(* Logix 5000 project; controller HP_SSC01 vendor 1 type 14 code 67 rev 17.7; software revision 17.01; part 8 of 15 *)
(* tags used below, declared in another part *)
   A_C3_0300 : ALIAS FOR C3_FaultStandard.0;
   A_C3_0301 : ALIAS FOR C3_FaultStandard.1;
   A_C3_0302 : ALIAS FOR C3_FaultStandard.2;
   A_C3_0303 : ALIAS FOR C3_FaultStandard.3;
   A_C3_0305 : ALIAS FOR C3_FaultStandard.5;
   A_C3_0309 : ALIAS FOR C3_FaultStandard.9;
   A_C3_0310 : ALIAS FOR C3_FaultStandard.10;
   A_C3_0311 : ALIAS FOR C3_FaultStandard.11;
   A_C3_0312 : ALIAS FOR C3_FaultStandard.12;
   A_C3_0313 : ALIAS FOR C3_FaultStandard.13;
   A_C3_0314 : ALIAS FOR C3_FaultStandard.14;
   A_C3_0315 : ALIAS FOR C3_FaultStandard.15;
   A_C3_0317 : ALIAS FOR C3_FaultStandard.17;
   A_C3_0319 : ALIAS FOR C3_FaultStandard.19;
   A_C3_0321 : ALIAS FOR C3_FaultStandard.21;
   A_C3_0322 : ALIAS FOR C3_FaultStandard.22;
   A_C3_0323 : ALIAS FOR C3_FaultStandard.23;
   A_C3_0324 : ALIAS FOR C3_FaultStandard.24;
   A_C3_0325 : ALIAS FOR C3_FaultStandard.25;
   A_C3_0327 : ALIAS FOR C3_FaultStandard.27;
   A_C3_0328 : ALIAS FOR C3_FaultStandard.28;
   A_C3_0329 : ALIAS FOR C3_FaultStandard.29;
   A_C3_0330 : ALIAS FOR C3_FaultStandard.30;
   A_C3_0331 : ALIAS FOR C3_FaultStandard.31;
   A_C3_0404 : ALIAS FOR C3_Warning.4;
   A_C3_0406 : ALIAS FOR C3_Warning.6;
   A_C3_0407 : ALIAS FOR C3_Warning.7;
   A_C3_0408 : ALIAS FOR C3_Warning.8;
   A_C3_0409 : ALIAS FOR C3_Warning.9;
   A_C3_0412 : ALIAS FOR C3_Warning.12;
   A_C3_0413 : ALIAS FOR C3_Warning.13;
   A_C3_0414 : ALIAS FOR C3_Warning.14;
   A_C3_0415 : ALIAS FOR C3_Warning.15;
   A_C3_0416 : ALIAS FOR C3_Warning.16;
   A_C3_0424 : ALIAS FOR C3_Warning.24;
   A_C3_0427 : ALIAS FOR C3_Warning.27;
   A_C3_0428 : ALIAS FOR C3_Warning.28;
   A_C3_0430 : ALIAS FOR C3_Warning.30;
   C3 : AXIS_SERVO_DRIVE;
   C3_32HourTimers : TIMER[4];
   C3_All_DLY_OK : BOOL;
   C3_BrakeSequenceInProcess : BOOL;
   C3_BrakeTest : BOOL;
   C3_BrakeTestEndPosition : REAL;
   C3_BrakeTestFailed : BOOL;
   C3_BrakeTestLocalDisable : BOOL;
   C3_BrakeTestMAJ01 : MOTION_INSTRUCTION;
   C3_BrakeTestMessageNumber : DINT;
   C3_BrakeTestONS : BOOL;
   C3_BrakeTestSelected : BOOL;
   C3_BrakeTestSequence : DINT;
   C3_BrakeTestSequenceAlarms : DINT;
   C3_BrakeTestSequenceAlarmTimer : TIMER[16];
   C3_BrakeTestSequenceONS : DINT;
   C3_BrakeTestStartPosition : REAL;
   C3_BrakeTestStoppingDistance : REAL;
   C3_BrakeTestTimerHoldVel : TIMER;
   C3_BrakeTestWarning : BOOL;
   C3_DisableTimer : TIMER;
   C3_DumpTest : BOOL;
   C3_DumpValveFailedOff : BOOL;
   C3_DumpValveFailedOn : BOOL;
   C3_DumpValveMessageNumber : DINT;
   C3_DumpValveTestDelay : TIMER[8];
   C3_DumpValveTestDelay2 : TIMER;
   C3_DumpValveTestSelected : BOOL;
   C3_DumpValveTestSequence : DINT;
   C3_DumpValveTestSequenceAlarms : DINT;
   C3_DumpValveTestSequenceAlarmTimer : TIMER[16];
   C3_EncoderCounts : DINT;
   C3_EncoderCountsRaw : ALIAS FOR C3_RIO_AENT:3:I.PresentData;
   C3_EncoderDegree : REAL;
   C3_FaultDebounce : TIMER[8];
   C3_FaultHoldTimer : TIMER[4];
   C3_FaultHomeSwitchNotFound : BOOL;
   C3_FaultStandard : DINT;
   C3_HomeInputStatus : BOOL;
   C3_HomeSequence : DINT;
   C3_HomeSequenceAlarms : DINT;
   C3_HomeSwitchFaultK7KFailedOff : BOOL;
   C3_HomeSwitchFaultK7KFailedOn : BOOL;
   C3_HomeSwitchFaultSafeFailedOff : BOOL;
   C3_HomeSwitchFaultSafeFailedOn : BOOL;
   C3_IndexEnable : BOOL;
   C3_JogEnable : BOOL;
   C3_LIM_ALARM_B : ALIAS FOR C3_RIO_AENT:I.Data[1].0;
   C3_MaintEnable : BOOL;
   C3_MotorActualPositionX1000 : DINT;
   C3_MotorAverageVelocityX1000 : DINT;
   C3_MotorFan : ALIAS FOR C3_RIO_AENT:O.Data[2].0;
   C3_MSF : MOTION_INSTRUCTION;
   C3_MSO : MOTION_INSTRUCTION;
   C3_OIT_Current : DINT;
   C3_ONS_Fault : DINT;
   C3_RemoteBrakeAndHomeSequenceAlarms : DINT;
   C3_RemoteBrakeTestCMD : BOOL;
   C3_RemoteDumpTestCMD : BOOL;
   C3_ServoActionStatusOffDelay : TIMER;
   C3_ServoActionStatusOnDelay : TIMER;
   C3_ServoFanOverload : ALIAS FOR C3_RIO_AENT:I.Data[1].2;
   C3_SS_LocalRemote_1_IsRemote : ALIAS FOR C3_RIO_AENT:1:I.3;
   C3_SS_RemoteMode : BOOL;
   C3_Warning : DINT;
   C3DumpValveTestSequenceONS : DINT;
   RCS_CMD_RunInAuto : BOOL;
   RCS_SyncMotionEnable : BOOL;
   S_C3_EncoderDegree : DINT;
   S_C3_ExecutePB : BOOL;
   S_C3_FaultReset : BOOL;
   S_C3_ModeLocal : BOOL;
   S_C3_ModeRemote : BOOL;
   S_C3_MotionEnabled : BOOL;
   S_C3_MSTOP_InputOK : BOOL;
   S_C3_NearOnPath : BOOL;
   S_C3_OffPath : BOOL;
   S_C3_OIT_FaultReset : BOOL;
   S_C3_OutputEnable : BOOL;
   S_C3_PressureOK : ALIAS FOR C3_Safe:I.Pt05Data;
   S_C3_SAFETY_ENABLE_1 : ALIAS FOR C3_Safe:O.Pt00Data;
   S_C3_SAFETY_ENABLE_2 : ALIAS FOR C3_Safe:O.Pt01Data;
   S_C3_Stop1_OK : BOOL;
   S_RCS_CMD_FaultReset : BOOL;
   STS_Enable_Rail : DINT;
   ZZZ_DIAG_A_C3_0302 : BOOL;
   ZZZ_DIAG_C3_AxisFault : DINT;
   ZZZ_DIAG_C3_AxisStatus : DINT;
   ZZZ_DIAG_C3_EnableRail : DINT;
   ZZZ_DIAG_C3_MotionStatus : DINT;
   ZZZ_DIAG_C3_MSF : MOTION_INSTRUCTION;
   ZZZ_DIAG_C3_MSO : MOTION_INSTRUCTION;
   ZZZ_DIAG_C3_OneTimeOnly : BOOL;
   ZZZ_DIAG_C3_OutputEnable : BOOL;
   ZZZ_DIAG_C3_OutputEnable_ACC : DINT;
   ZZZ_DIAG_ONS : DINT;
   ZZZ_DIAG_S_C3_OutputEnableTON : TIMER;
   ZZZ_DIAG_S_C3_SAFETY_ENABLE_1 : BOOL;
   ZZZ_DIAG_S_C3_SAFETY_ENABLE_2 : BOOL;

PROGRAM Carousel3   (* main routine C300_Main *)
VAR
   zzz_Test30 : BOOL;
   zzz_Test31 : BOOL;
END_VAR

ROUTINE C300_Main   (* ladder *)
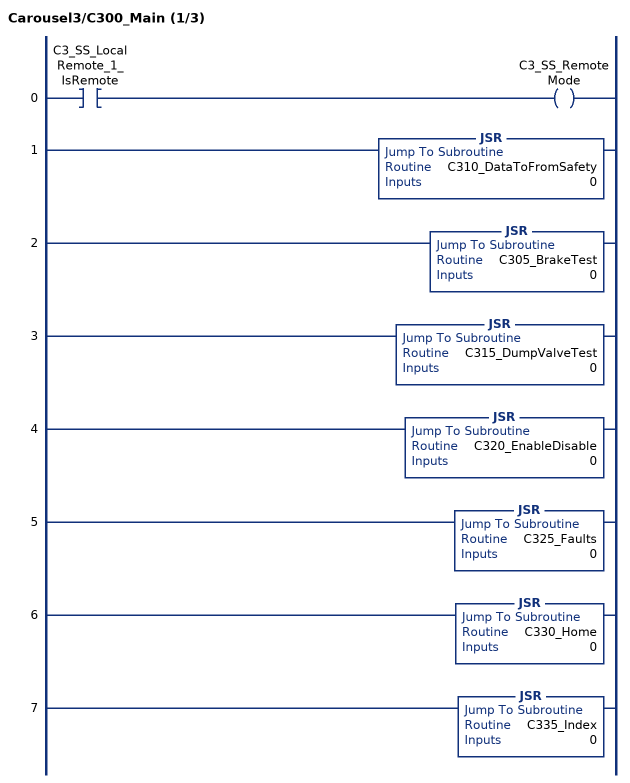
   0: XIC(C3_SS_LocalRemote_1_IsRemote)OTE(C3_SS_RemoteMode);
   1: JSR(C310_DataToFromSafety,0);
   2: JSR(C305_BrakeTest,0);
   3: JSR(C315_DumpValveTest,0);
   4: JSR(C320_EnableDisable,0);
   5: JSR(C325_Faults,0);
   6: JSR(C330_Home,0);
   7: JSR(C335_Index,0);
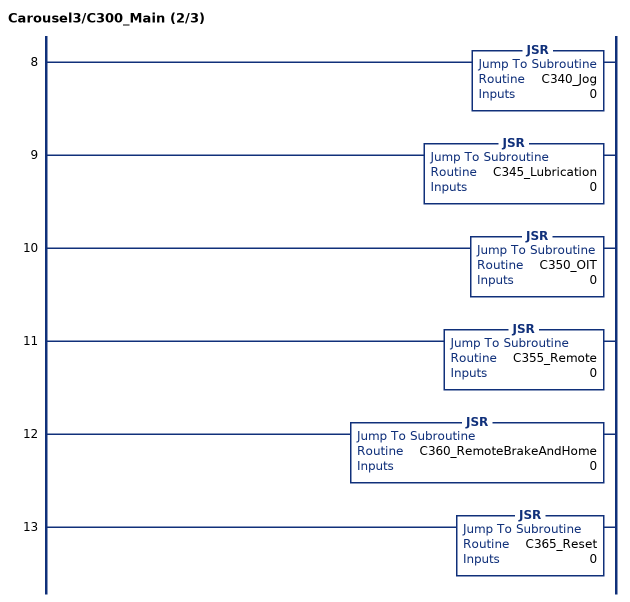
   8: JSR(C340_Jog,0);
   9: JSR(C345_Lubrication,0);
   10: JSR(C350_OIT,0);
   11: JSR(C355_Remote,0);
   12: JSR(C360_RemoteBrakeAndHome,0);
   13: JSR(C365_Reset,0);
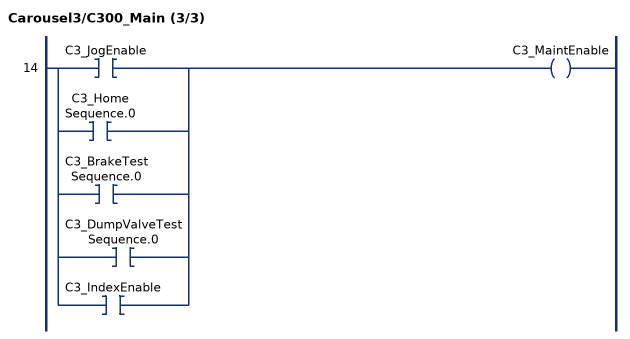
   14: [XIC(C3_JogEnable) ,XIC(C3_HomeSequence.0) ,XIC(C3_BrakeTestSequence.0) ,XIC(C3_DumpValveTestSequence.0) ,XIC(C3_IndexEnable) ]OTE(C3_MaintEnable);
END_ROUTINE

ROUTINE C305_BrakeTest   (* ladder *)
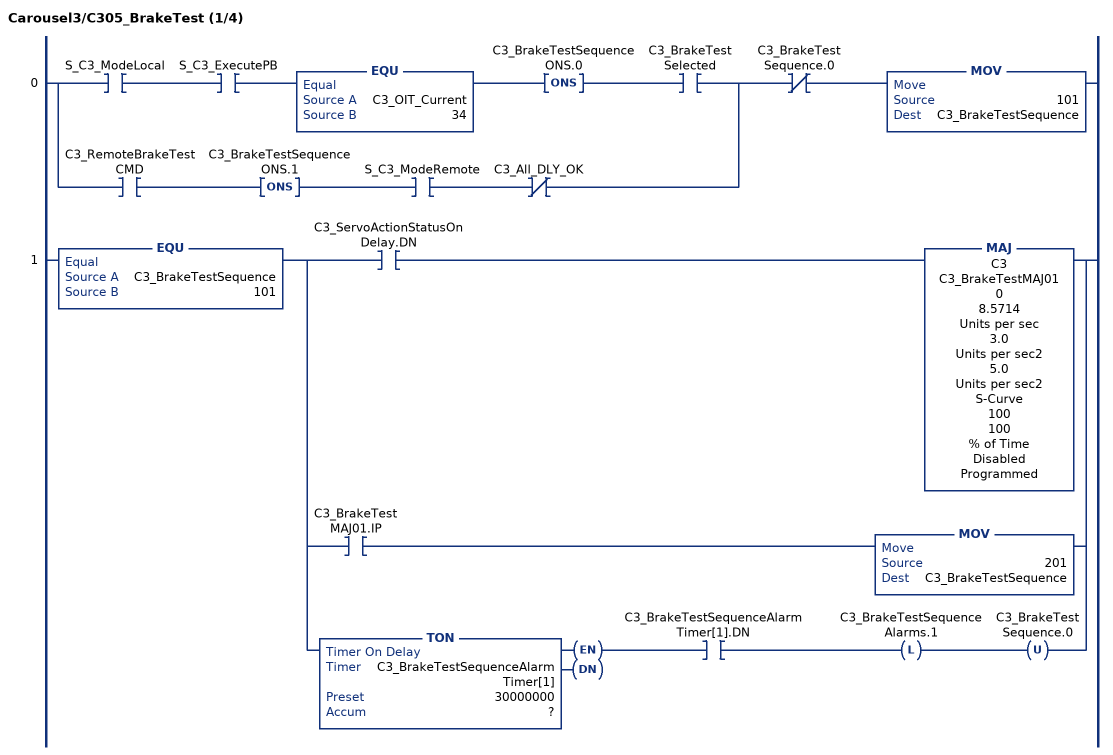
   0: [XIC(S_C3_ModeLocal) XIC(S_C3_ExecutePB) EQU(C3_OIT_Current,34) ONS(C3_BrakeTestSequenceONS.0) XIC(C3_BrakeTestSelected) ,XIC(C3_RemoteBrakeTestCMD) ONS(C3_BrakeTestSequenceONS.1) XIC(S_C3_ModeRemote) XIO(C3_All_DLY_OK) ]XIO(C3_BrakeTestSequence.0)MOV(101,C3_BrakeTestSequence);
   1: EQU(C3_BrakeTestSequence,101)[XIC(C3_ServoActionStatusOnDelay.DN) MAJ(C3,C3_BrakeTestMAJ01,0,8.5714,Units per sec,3.0,Units per sec2,5.0,Units per sec2,S-Curve,100,100,% of Time,Disabled,Programmed) ,XIC(C3_BrakeTestMAJ01.IP) MOV(201,C3_BrakeTestSequence) ,TON(C3_BrakeTestSequenceAlarmTimer[1],?,?) XIC(C3_BrakeTestSequenceAlarmTimer[1].DN) OTL(C3_BrakeTestSequenceAlarms.1) OTU(C3_BrakeTestSequence.0) ];
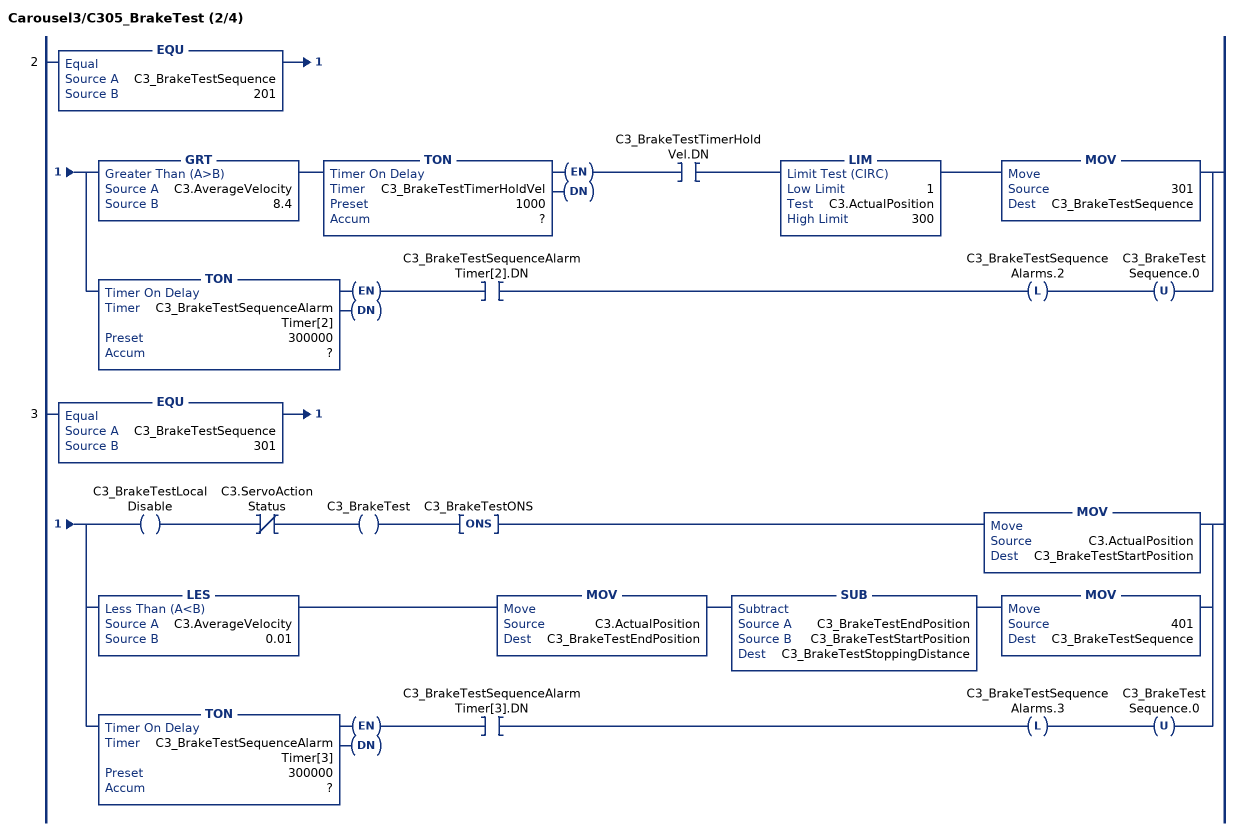
   2: EQU(C3_BrakeTestSequence,201)[GRT(C3.AverageVelocity,8.4) TON(C3_BrakeTestTimerHoldVel,?,?) XIC(C3_BrakeTestTimerHoldVel.DN) LIM(1,C3.ActualPosition,300) MOV(301,C3_BrakeTestSequence) ,TON(C3_BrakeTestSequenceAlarmTimer[2],?,?) XIC(C3_BrakeTestSequenceAlarmTimer[2].DN) OTL(C3_BrakeTestSequenceAlarms.2) OTU(C3_BrakeTestSequence.0) ];
   3: EQU(C3_BrakeTestSequence,301)[OTE(C3_BrakeTestLocalDisable) XIO(C3.ServoActionStatus) OTE(C3_BrakeTest) ONS(C3_BrakeTestONS) MOV(C3.ActualPosition,C3_BrakeTestStartPosition) ,LES(C3.AverageVelocity,0.01) MOV(C3.ActualPosition,C3_BrakeTestEndPosition) SUB(C3_BrakeTestEndPosition,C3_BrakeTestStartPosition,C3_BrakeTestStoppingDistance) MOV(401,C3_BrakeTestSequence) ,TON(C3_BrakeTestSequenceAlarmTimer[3],?,?) XIC(C3_BrakeTestSequenceAlarmTimer[3].DN) OTL(C3_BrakeTestSequenceAlarms.3) OTU(C3_BrakeTestSequence.0) ];
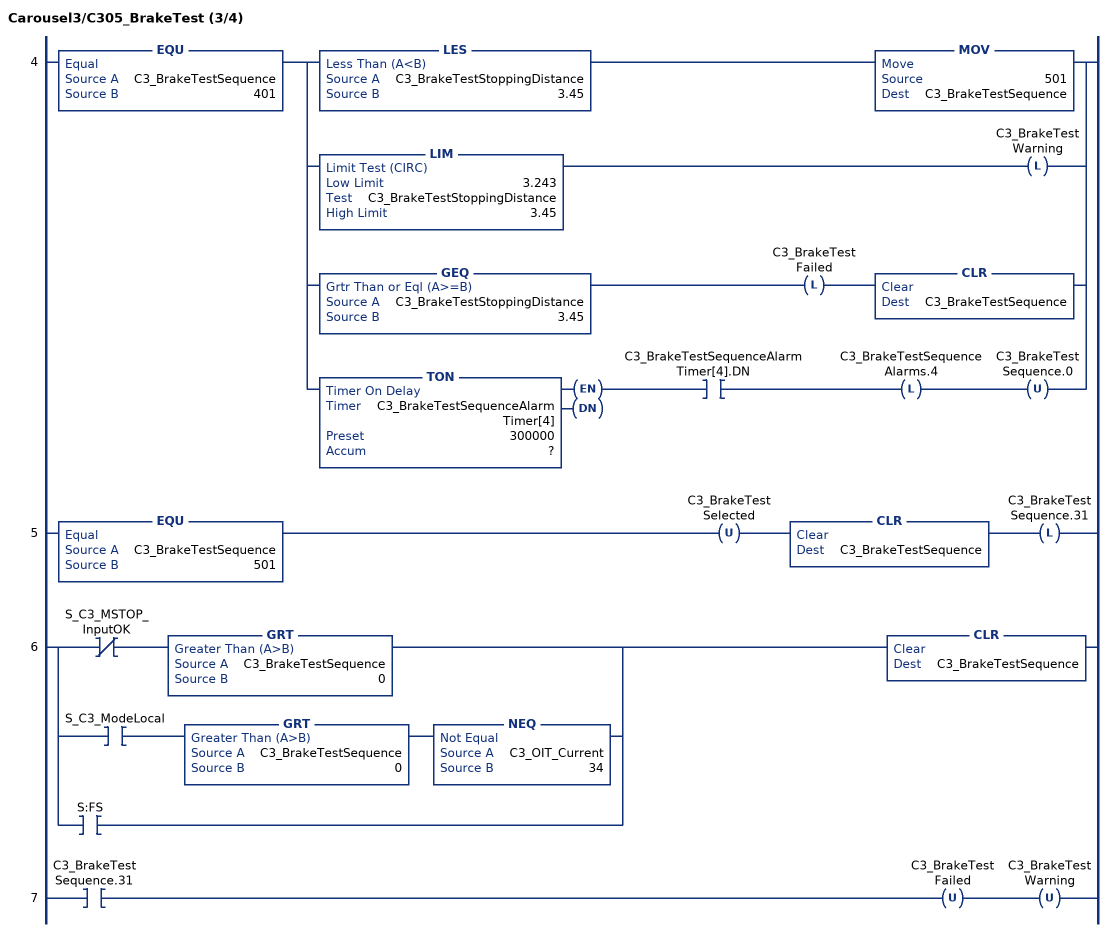
   4: EQU(C3_BrakeTestSequence,401)[LES(C3_BrakeTestStoppingDistance,3.45) MOV(501,C3_BrakeTestSequence) ,LIM(3.243,C3_BrakeTestStoppingDistance,3.45) OTL(C3_BrakeTestWarning) ,GEQ(C3_BrakeTestStoppingDistance,3.45) OTL(C3_BrakeTestFailed) CLR(C3_BrakeTestSequence) ,TON(C3_BrakeTestSequenceAlarmTimer[4],?,?) XIC(C3_BrakeTestSequenceAlarmTimer[4].DN) OTL(C3_BrakeTestSequenceAlarms.4) OTU(C3_BrakeTestSequence.0) ];
   5: EQU(C3_BrakeTestSequence,501)OTU(C3_BrakeTestSelected)CLR(C3_BrakeTestSequence)OTL(C3_BrakeTestSequence.31);
   6: [XIO(S_C3_MSTOP_InputOK) GRT(C3_BrakeTestSequence,0) ,XIC(S_C3_ModeLocal) GRT(C3_BrakeTestSequence,0) NEQ(C3_OIT_Current,34) ,XIC(S:FS) ]CLR(C3_BrakeTestSequence);
   7: XIC(C3_BrakeTestSequence.31)OTU(C3_BrakeTestFailed)OTU(C3_BrakeTestWarning);
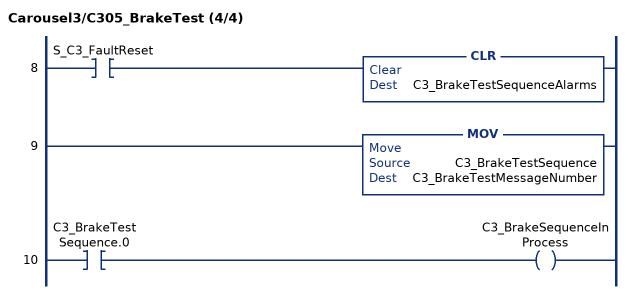
   8: XIC(S_C3_FaultReset)CLR(C3_BrakeTestSequenceAlarms);
   9: MOV(C3_BrakeTestSequence,C3_BrakeTestMessageNumber);
   10: XIC(C3_BrakeTestSequence.0)OTE(C3_BrakeSequenceInProcess);
END_ROUTINE

ROUTINE C310_DataToFromSafety   (* ladder *)
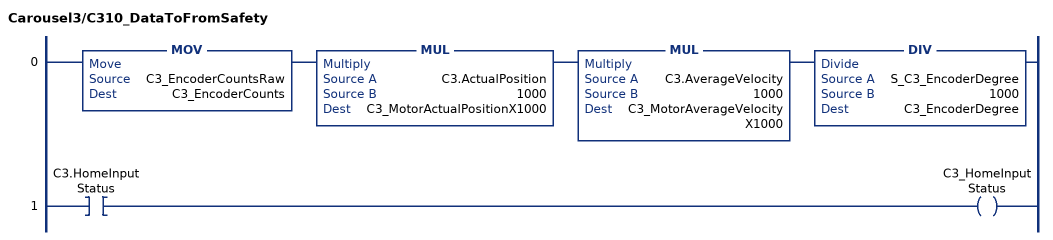
   0: MOV(C3_EncoderCountsRaw,C3_EncoderCounts)MUL(C3.ActualPosition,1000,C3_MotorActualPositionX1000)MUL(C3.AverageVelocity,1000,C3_MotorAverageVelocityX1000)DIV(S_C3_EncoderDegree,1000,C3_EncoderDegree);
   1: XIC(C3.HomeInputStatus)OTE(C3_HomeInputStatus);
END_ROUTINE

ROUTINE C315_DumpValveTest   (* ladder *)
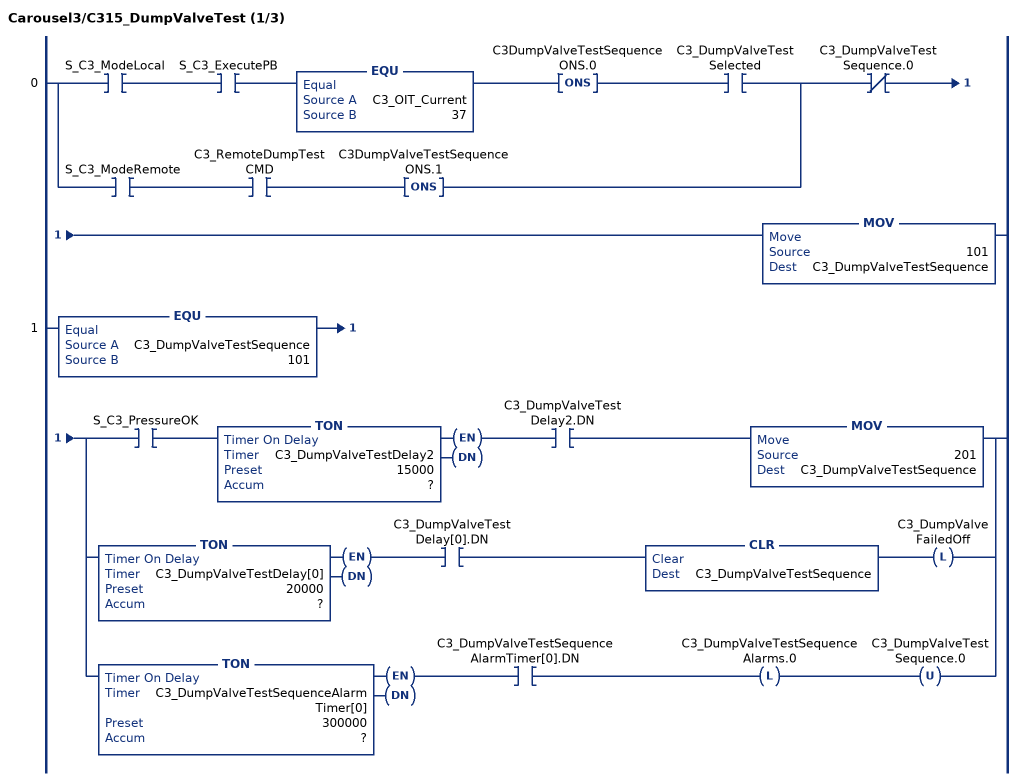
   0: [XIC(S_C3_ModeLocal) XIC(S_C3_ExecutePB) EQU(C3_OIT_Current,37) ONS(C3DumpValveTestSequenceONS.0) XIC(C3_DumpValveTestSelected) ,XIC(S_C3_ModeRemote) XIC(C3_RemoteDumpTestCMD) ONS(C3DumpValveTestSequenceONS.1) ]XIO(C3_DumpValveTestSequence.0)MOV(101,C3_DumpValveTestSequence);
   1: EQU(C3_DumpValveTestSequence,101)[XIC(S_C3_PressureOK) TON(C3_DumpValveTestDelay2,?,?) XIC(C3_DumpValveTestDelay2.DN) MOV(201,C3_DumpValveTestSequence) ,TON(C3_DumpValveTestDelay[0],?,?) XIC(C3_DumpValveTestDelay[0].DN) CLR(C3_DumpValveTestSequence) OTL(C3_DumpValveFailedOff) ,TON(C3_DumpValveTestSequenceAlarmTimer[0],?,?) XIC(C3_DumpValveTestSequenceAlarmTimer[0].DN) OTL(C3_DumpValveTestSequenceAlarms.0) OTU(C3_DumpValveTestSequence.0) ];
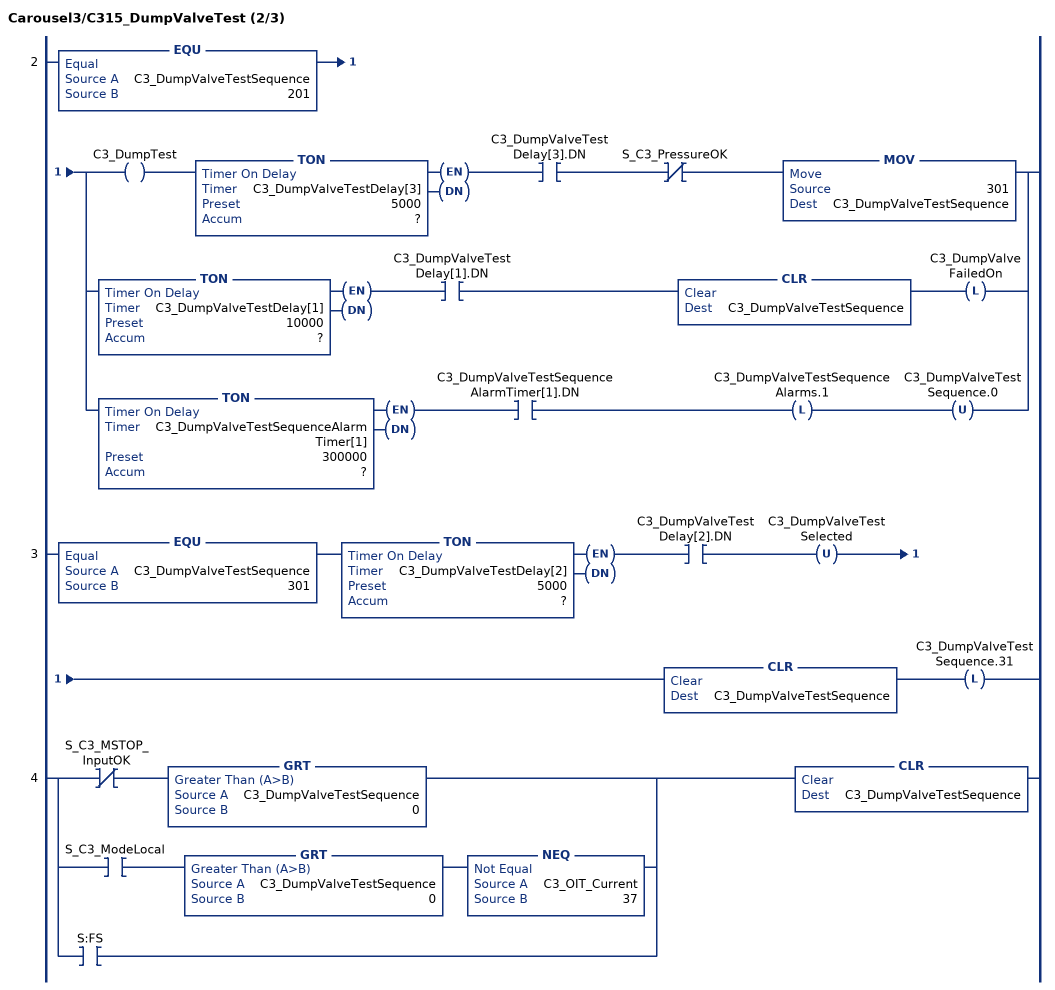
   2: EQU(C3_DumpValveTestSequence,201)[OTE(C3_DumpTest) TON(C3_DumpValveTestDelay[3],?,?) XIC(C3_DumpValveTestDelay[3].DN) XIO(S_C3_PressureOK) MOV(301,C3_DumpValveTestSequence) ,TON(C3_DumpValveTestDelay[1],?,?) XIC(C3_DumpValveTestDelay[1].DN) CLR(C3_DumpValveTestSequence) OTL(C3_DumpValveFailedOn) ,TON(C3_DumpValveTestSequenceAlarmTimer[1],?,?) XIC(C3_DumpValveTestSequenceAlarmTimer[1].DN) OTL(C3_DumpValveTestSequenceAlarms.1) OTU(C3_DumpValveTestSequence.0) ];
   3: EQU(C3_DumpValveTestSequence,301)TON(C3_DumpValveTestDelay[2],?,?)XIC(C3_DumpValveTestDelay[2].DN)OTU(C3_DumpValveTestSelected)CLR(C3_DumpValveTestSequence)OTL(C3_DumpValveTestSequence.31);
   4: [XIO(S_C3_MSTOP_InputOK) GRT(C3_DumpValveTestSequence,0) ,XIC(S_C3_ModeLocal) GRT(C3_DumpValveTestSequence,0) NEQ(C3_OIT_Current,37) ,XIC(S:FS) ]CLR(C3_DumpValveTestSequence);
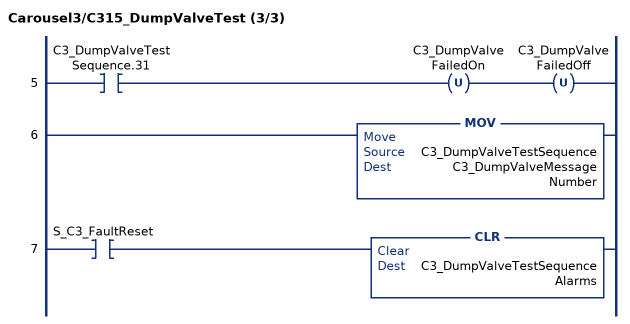
   5: XIC(C3_DumpValveTestSequence.31)OTU(C3_DumpValveFailedOn)OTU(C3_DumpValveFailedOff);
   6: MOV(C3_DumpValveTestSequence,C3_DumpValveMessageNumber);
   7: XIC(S_C3_FaultReset)CLR(C3_DumpValveTestSequenceAlarms);
END_ROUTINE

ROUTINE C320_EnableDisable   (* ladder *)
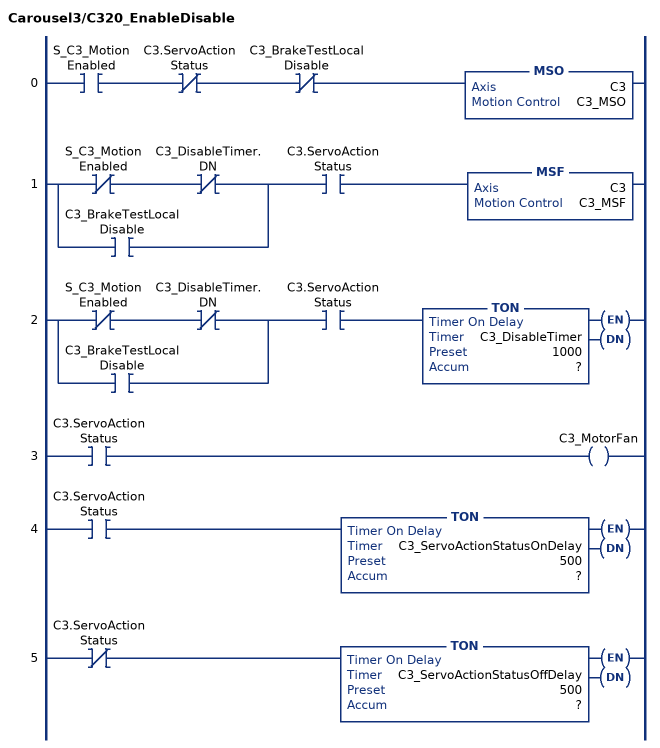
   0: XIC(S_C3_MotionEnabled)XIO(C3.ServoActionStatus)XIO(C3_BrakeTestLocalDisable)MSO(C3,C3_MSO);
   1: [XIO(S_C3_MotionEnabled) XIO(C3_DisableTimer.DN) ,XIC(C3_BrakeTestLocalDisable) ]XIC(C3.ServoActionStatus)MSF(C3,C3_MSF);
   2: [XIO(S_C3_MotionEnabled) XIO(C3_DisableTimer.DN) ,XIC(C3_BrakeTestLocalDisable) ]XIC(C3.ServoActionStatus)TON(C3_DisableTimer,?,?);
   3: XIC(C3.ServoActionStatus)OTE(C3_MotorFan);
   4: XIC(C3.ServoActionStatus)TON(C3_ServoActionStatusOnDelay,?,?);
   5: XIO(C3.ServoActionStatus)TON(C3_ServoActionStatusOffDelay,?,?);
END_ROUTINE

ROUTINE C325_Faults   (* ladder *)
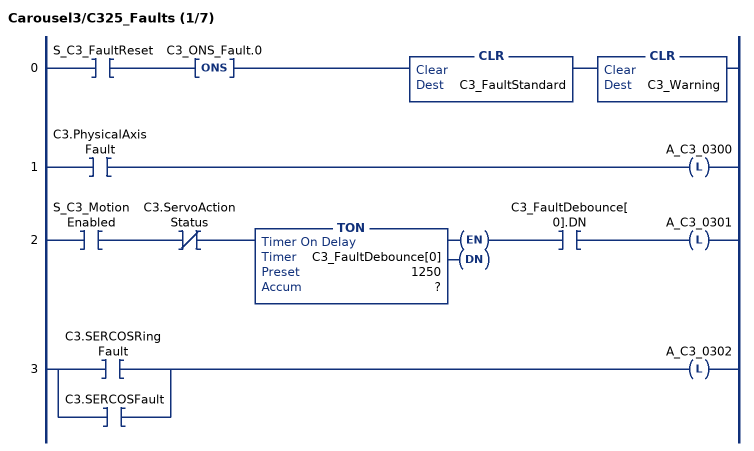
   0: XIC(S_C3_FaultReset)ONS(C3_ONS_Fault.0)CLR(C3_FaultStandard)CLR(C3_Warning);
   1: XIC(C3.PhysicalAxisFault)OTL(A_C3_0300);
   2: XIC(S_C3_MotionEnabled)XIO(C3.ServoActionStatus)TON(C3_FaultDebounce[0],?,?)XIC(C3_FaultDebounce[0].DN)OTL(A_C3_0301);
   3: [XIC(C3.SERCOSRingFault) ,XIC(C3.SERCOSFault) ]OTL(A_C3_0302);
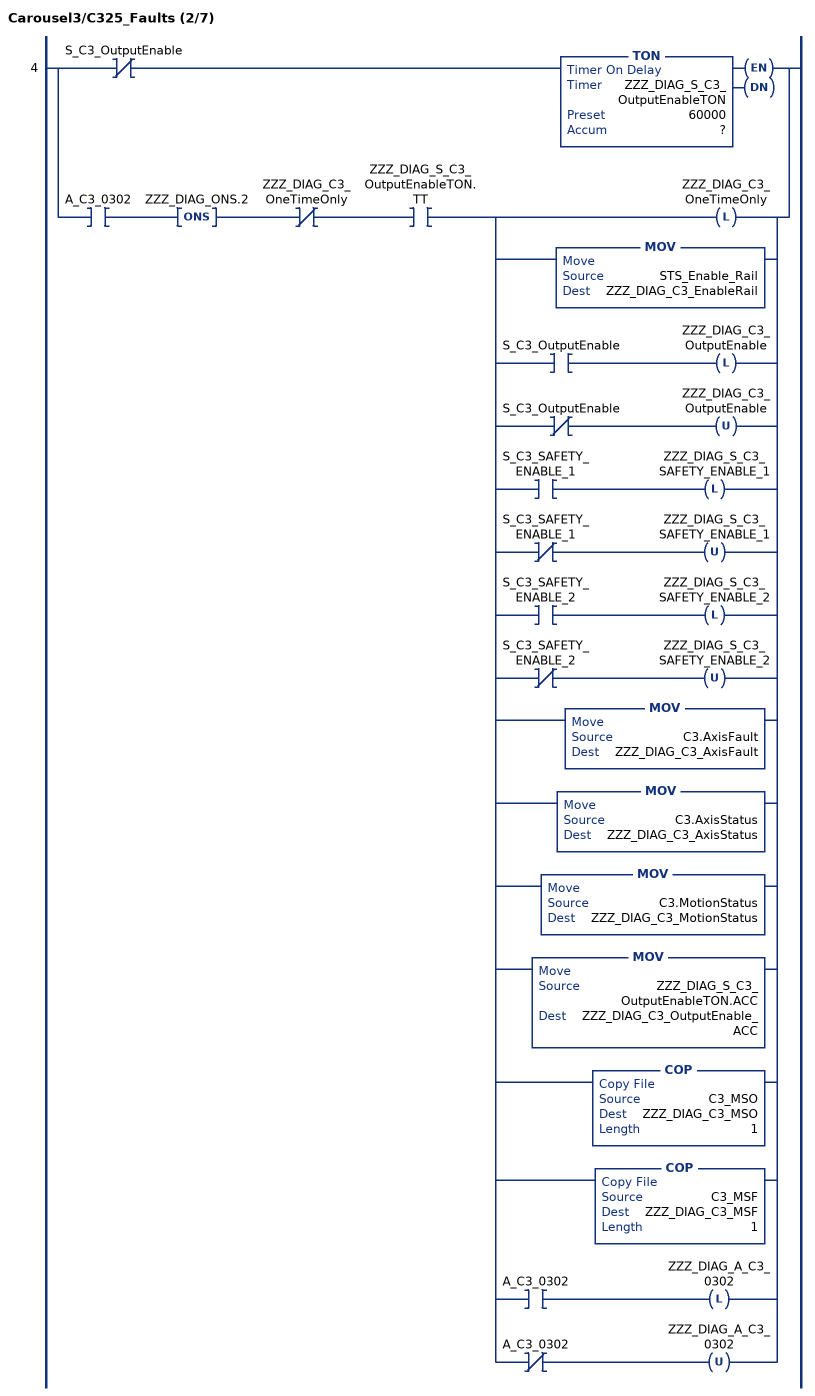
   4: [XIO(S_C3_OutputEnable) TON(ZZZ_DIAG_S_C3_OutputEnableTON,?,?) ,XIC(A_C3_0302) ONS(ZZZ_DIAG_ONS.2) XIO(ZZZ_DIAG_C3_OneTimeOnly) XIC(ZZZ_DIAG_S_C3_OutputEnableTON.TT) [OTL(ZZZ_DIAG_C3_OneTimeOnly) ,MOV(STS_Enable_Rail,ZZZ_DIAG_C3_EnableRail) ,XIC(S_C3_OutputEnable) OTL(ZZZ_DIAG_C3_OutputEnable) ,XIO(S_C3_OutputEnable) OTU(ZZZ_DIAG_C3_OutputEnable) ,XIC(S_C3_SAFETY_ENABLE_1) OTL(ZZZ_DIAG_S_C3_SAFETY_ENABLE_1) ,XIO(S_C3_SAFETY_ENABLE_1) OTU(ZZZ_DIAG_S_C3_SAFETY_ENABLE_1) ,XIC(S_C3_SAFETY_ENABLE_2) OTL(ZZZ_DIAG_S_C3_SAFETY_ENABLE_2) ,XIO(S_C3_SAFETY_ENABLE_2) OTU(ZZZ_DIAG_S_C3_SAFETY_ENABLE_2) ,MOV(C3.AxisFault,ZZZ_DIAG_C3_AxisFault) ,MOV(C3.AxisStatus,ZZZ_DIAG_C3_AxisStatus) ,MOV(C3.MotionStatus,ZZZ_DIAG_C3_MotionStatus) ,MOV(ZZZ_DIAG_S_C3_OutputEnableTON.ACC,ZZZ_DIAG_C3_OutputEnable_ACC) ,COP(C3_MSO,ZZZ_DIAG_C3_MSO,1) ,COP(C3_MSF,ZZZ_DIAG_C3_MSF,1) ,XIC(A_C3_0302) OTL(ZZZ_DIAG_A_C3_0302) ,XIO(A_C3_0302) OTU(ZZZ_DIAG_A_C3_0302) ] ];
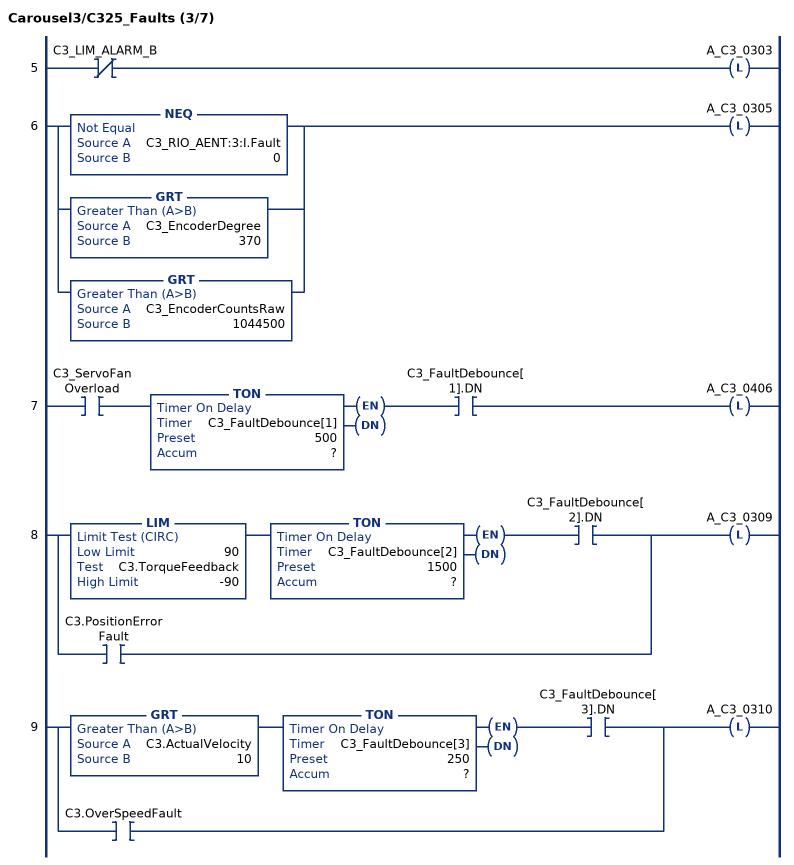
   5: XIO(C3_LIM_ALARM_B)OTL(A_C3_0303);
   6: [NEQ(C3_RIO_AENT:3:I.Fault,0) ,GRT(C3_EncoderDegree,370) ,GRT(C3_EncoderCountsRaw,1044500) ]OTL(A_C3_0305);
   7: XIC(C3_ServoFanOverload)TON(C3_FaultDebounce[1],?,?)XIC(C3_FaultDebounce[1].DN)OTL(A_C3_0406);
   8: [LIM(90,C3.TorqueFeedback,-90) TON(C3_FaultDebounce[2],?,?) XIC(C3_FaultDebounce[2].DN) ,XIC(C3.PositionErrorFault) ]OTL(A_C3_0309);
   9: [GRT(C3.ActualVelocity,10) TON(C3_FaultDebounce[3],?,?) XIC(C3_FaultDebounce[3].DN) ,XIC(C3.OverSpeedFault) ]OTL(A_C3_0310);
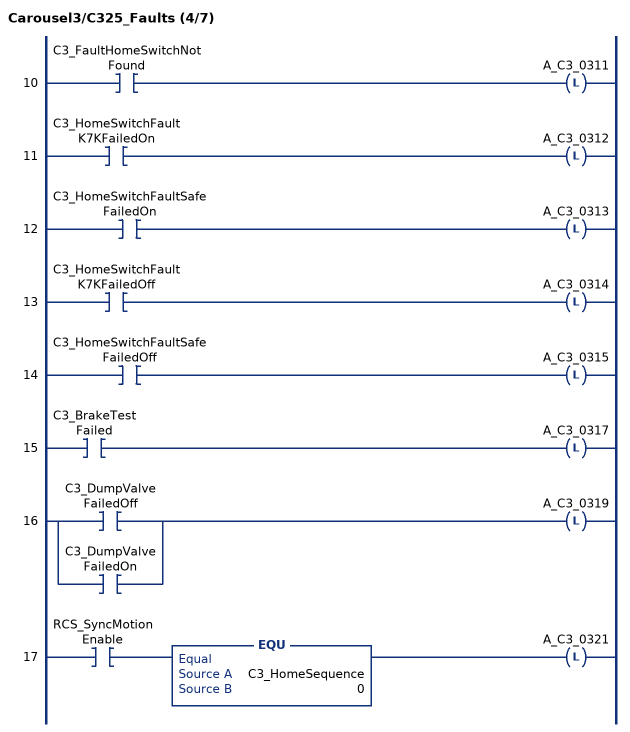
   10: XIC(C3_FaultHomeSwitchNotFound)OTL(A_C3_0311);
   11: XIC(C3_HomeSwitchFaultK7KFailedOn)OTL(A_C3_0312);
   12: XIC(C3_HomeSwitchFaultSafeFailedOn)OTL(A_C3_0313);
   13: XIC(C3_HomeSwitchFaultK7KFailedOff)OTL(A_C3_0314);
   14: XIC(C3_HomeSwitchFaultSafeFailedOff)OTL(A_C3_0315);
   15: XIC(C3_BrakeTestFailed)OTL(A_C3_0317);
   16: [XIC(C3_DumpValveFailedOff) ,XIC(C3_DumpValveFailedOn) ]OTL(A_C3_0319);
   17: XIC(RCS_SyncMotionEnable)EQU(C3_HomeSequence,0)OTL(A_C3_0321);
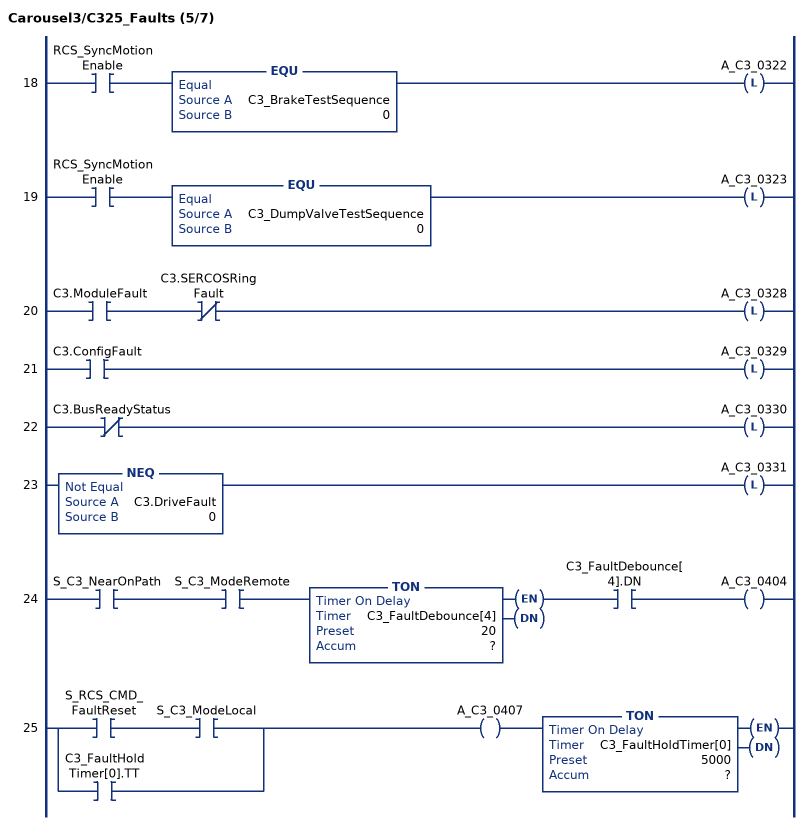
   18: XIC(RCS_SyncMotionEnable)EQU(C3_BrakeTestSequence,0)OTL(A_C3_0322);
   19: XIC(RCS_SyncMotionEnable)EQU(C3_DumpValveTestSequence,0)OTL(A_C3_0323);
   20: XIC(C3.ModuleFault)XIO(C3.SERCOSRingFault)OTL(A_C3_0328);
   21: XIC(C3.ConfigFault)OTL(A_C3_0329);
   22: XIO(C3.BusReadyStatus)OTL(A_C3_0330);
   23: NEQ(C3.DriveFault,0)OTL(A_C3_0331);
   24: XIC(S_C3_NearOnPath)XIC(S_C3_ModeRemote)TON(C3_FaultDebounce[4],?,?)XIC(C3_FaultDebounce[4].DN)OTE(A_C3_0404);
   25: [XIC(S_RCS_CMD_FaultReset) XIC(S_C3_ModeLocal) ,XIC(C3_FaultHoldTimer[0].TT) ]OTE(A_C3_0407)TON(C3_FaultHoldTimer[0],?,?);
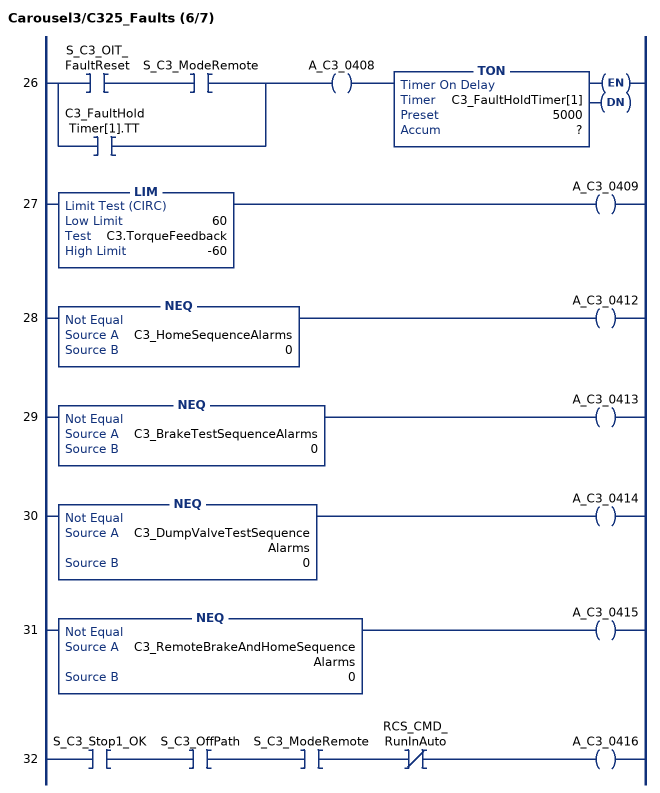
   26: [XIC(S_C3_OIT_FaultReset) XIC(S_C3_ModeRemote) ,XIC(C3_FaultHoldTimer[1].TT) ]OTE(A_C3_0408)TON(C3_FaultHoldTimer[1],?,?);
   27: LIM(60,C3.TorqueFeedback,-60)OTE(A_C3_0409);
   28: NEQ(C3_HomeSequenceAlarms,0)OTE(A_C3_0412);
   29: NEQ(C3_BrakeTestSequenceAlarms,0)OTE(A_C3_0413);
   30: NEQ(C3_DumpValveTestSequenceAlarms,0)OTE(A_C3_0414);
   31: NEQ(C3_RemoteBrakeAndHomeSequenceAlarms,0)OTE(A_C3_0415);
   32: XIC(S_C3_Stop1_OK)XIC(S_C3_OffPath)XIC(S_C3_ModeRemote)XIO(RCS_CMD_RunInAuto)OTE(A_C3_0416);
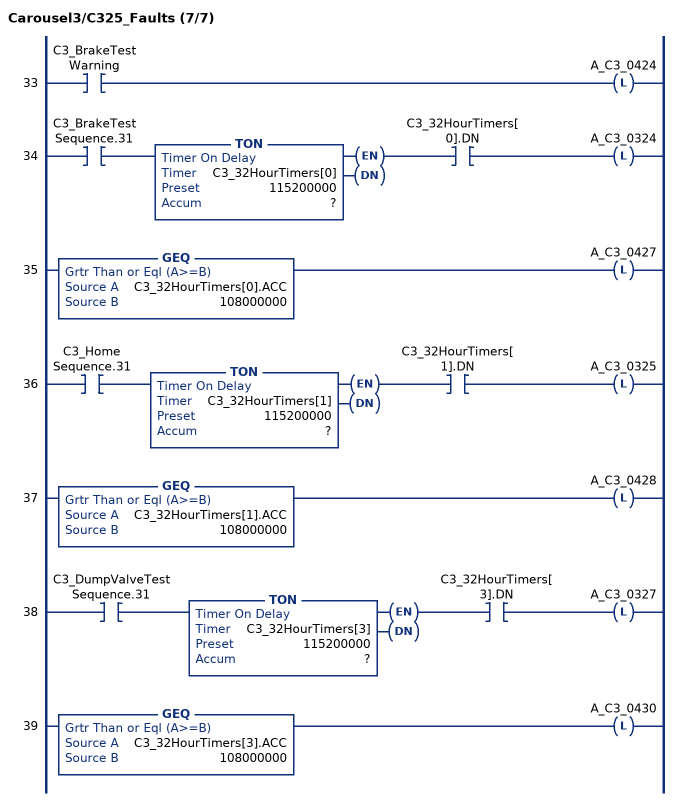
   33: XIC(C3_BrakeTestWarning)OTL(A_C3_0424);
   34: XIC(C3_BrakeTestSequence.31)TON(C3_32HourTimers[0],?,?)XIC(C3_32HourTimers[0].DN)OTL(A_C3_0324);
   35: GEQ(C3_32HourTimers[0].ACC,108000000)OTL(A_C3_0427);
   36: XIC(C3_HomeSequence.31)TON(C3_32HourTimers[1],?,?)XIC(C3_32HourTimers[1].DN)OTL(A_C3_0325);
   37: GEQ(C3_32HourTimers[1].ACC,108000000)OTL(A_C3_0428);
   38: XIC(C3_DumpValveTestSequence.31)TON(C3_32HourTimers[3],?,?)XIC(C3_32HourTimers[3].DN)OTL(A_C3_0327);
   39: GEQ(C3_32HourTimers[3].ACC,108000000)OTL(A_C3_0430);
END_ROUTINE
